(* IEC 61131-3 sources: plc-automation-skill/codesys-st, 4 files *)

(* ---- DUT_CascadeTypes.ST ---- *)
TYPE E_CascadeState :
(
    Stopped := 0,
    SelectLead := 10,
    StartLead := 20,
    RunningCascade := 30,
    StageUp := 40,
    StageDown := 50,
    Tripped := 90
);
END_TYPE

TYPE ST_VSD_Cmd :
STRUCT
    xInhibit : BOOL;
    xRunCmd : BOOL;
    rSpeedRefPct : REAL;
END_STRUCT
END_TYPE

TYPE ST_VSD_Sts :
STRUCT
    xReady : BOOL;
    xRunning : BOOL;
    xFaulted : BOOL;
    xLocal : BOOL;
    xAvailable : BOOL;
    xTripLatched : BOOL;
    xStartFail : BOOL;
    rRuntimeHours : REAL;
    rSpeedFbPct : REAL;
END_STRUCT
END_TYPE

TYPE ST_VSD :
STRUCT
    Cmd : ST_VSD_Cmd;
    Sts : ST_VSD_Sts;
END_STRUCT
END_TYPE

TYPE ST_CascadeCmd :
STRUCT
    xAutoMode : BOOL;
    xManualMode : BOOL;
    xStart : BOOL;
    xStop : BOOL;
    xReset : BOOL;
    xRotateLead : BOOL;
END_STRUCT
END_TYPE

TYPE ST_CascadeCfg :
STRUCT
    iMaxRunning : INT := 5;
    rStageOnSpeedPct : REAL := 90.0;
    rStageOffSpeedPct : REAL := 45.0;
    tStageOnDelay : TIME := T#30S;
    tStageOffDelay : TIME := T#60S;
    tStartTimeout : TIME := T#10S;
    tMinRunTime : TIME := T#120S;
    tMinStopTime : TIME := T#120S;
    rSpeedMinPct : REAL := 0.0;
    rSpeedMaxPct : REAL := 100.0;
END_STRUCT
END_TYPE

TYPE ST_CascadeSts :
STRUCT
    eState : E_CascadeState;
    xAnyTrip : BOOL;
    xPermissiveOK : BOOL;
    iRunningCount : INT;
    iAvailableCount : INT;
    iLeadIndex : INT;
    iNextStageIndex : INT;
    rSpeedDemandPct : REAL;
    xAlarmNoAvailableVSD : BOOL;
    xAlarmStageFail : BOOL;
END_STRUCT
END_TYPE

TYPE ST_Cascade :
STRUCT
    Cmd : ST_CascadeCmd;
    Cfg : ST_CascadeCfg;
    Sts : ST_CascadeSts;
    rPV : REAL;
    rSP : REAL;
    rPIDOutPct : REAL;
END_STRUCT
END_TYPE

(* ---- GVL_IO.ST ---- *)
VAR_GLOBAL
    (* Group control and status. Bind HMI/SCADA tags to CP01 where required. *)
    CP01 : ST_Cascade;

    (* Internal VSD array, indexes 1..5. *)
    CP01_VSD : ARRAY[1..5] OF ST_VSD;

    (* Safety/process permissives mapped from real I/O or safety status. *)
    CP01_xEStopOK : BOOL;
    CP01_xProcessPermissiveOK : BOOL;

    (* Raw VSD inputs. Replace these with mapped fieldbus or I/O addresses. *)
    I_VSD01_xReady : BOOL;
    I_VSD01_xRunning : BOOL;
    I_VSD01_xFaulted : BOOL;
    I_VSD01_xLocal : BOOL;

    I_VSD02_xReady : BOOL;
    I_VSD02_xRunning : BOOL;
    I_VSD02_xFaulted : BOOL;
    I_VSD02_xLocal : BOOL;

    I_VSD03_xReady : BOOL;
    I_VSD03_xRunning : BOOL;
    I_VSD03_xFaulted : BOOL;
    I_VSD03_xLocal : BOOL;

    I_VSD04_xReady : BOOL;
    I_VSD04_xRunning : BOOL;
    I_VSD04_xFaulted : BOOL;
    I_VSD04_xLocal : BOOL;

    I_VSD05_xReady : BOOL;
    I_VSD05_xRunning : BOOL;
    I_VSD05_xFaulted : BOOL;
    I_VSD05_xLocal : BOOL;

    (* Raw VSD outputs. Replace these with mapped fieldbus or I/O addresses. *)
    O_VSD01_xRunCmd : BOOL;
    O_VSD01_rSpeedRefPct : REAL;

    O_VSD02_xRunCmd : BOOL;
    O_VSD02_rSpeedRefPct : REAL;

    O_VSD03_xRunCmd : BOOL;
    O_VSD03_rSpeedRefPct : REAL;

    O_VSD04_xRunCmd : BOOL;
    O_VSD04_rSpeedRefPct : REAL;

    O_VSD05_xRunCmd : BOOL;
    O_VSD05_rSpeedRefPct : REAL;
END_VAR

(* ---- FB_VSD_Cascade5.ST ---- *)
FUNCTION_BLOCK FB_VSD_Cascade5
VAR_INPUT
    xEStopOK : BOOL;
    xProcessPermissiveOK : BOOL;
    stCmd : ST_CascadeCmd;
    stCfg : ST_CascadeCfg;
    rPIDOutPct : REAL;
END_VAR
VAR_IN_OUT
    aVSD : ARRAY[1..5] OF ST_VSD;
END_VAR
VAR_OUTPUT
    stSts : ST_CascadeSts;
END_VAR
VAR
    i : INT;
    iScanIndex : INT;
    iNextLeadIndex : INT := 1;
    xRotateLeadPrev : BOOL;
    tStageOn : TON;
    tStageOff : TON;
    atStartFail : ARRAY[1..5] OF TON;
    atMinRun : ARRAY[1..5] OF TON;
    atMinStop : ARRAY[1..5] OF TON;
    cfg : ST_CascadeCfg;
END_VAR

(* Clamp configuration locally. *)
cfg := stCfg;

IF cfg.iMaxRunning < 1 THEN
    cfg.iMaxRunning := 1;
ELSIF cfg.iMaxRunning > 5 THEN
    cfg.iMaxRunning := 5;
END_IF;

IF cfg.rSpeedMinPct < 0.0 THEN
    cfg.rSpeedMinPct := 0.0;
END_IF;

IF cfg.rSpeedMaxPct > 100.0 THEN
    cfg.rSpeedMaxPct := 100.0;
END_IF;

IF cfg.rSpeedMaxPct < cfg.rSpeedMinPct THEN
    cfg.rSpeedMaxPct := cfg.rSpeedMinPct;
END_IF;

(* Clamp speed demand. PID is normally calculated outside this FB. *)
stSts.rSpeedDemandPct := rPIDOutPct;
IF stSts.rSpeedDemandPct < cfg.rSpeedMinPct THEN
    stSts.rSpeedDemandPct := cfg.rSpeedMinPct;
ELSIF stSts.rSpeedDemandPct > cfg.rSpeedMaxPct THEN
    stSts.rSpeedDemandPct := cfg.rSpeedMaxPct;
END_IF;

(* Group permissive. Reset never starts equipment. *)
stSts.xPermissiveOK :=
    stCmd.xAutoMode AND
    xEStopOK AND
    xProcessPermissiveOK;

stSts.xAnyTrip := (NOT xEStopOK) OR (NOT xProcessPermissiveOK);

(* Rotate preferred lead for next start. *)
IF stCmd.xRotateLead AND NOT xRotateLeadPrev THEN
    iNextLeadIndex := iNextLeadIndex + 1;
    IF iNextLeadIndex > 5 THEN
        iNextLeadIndex := 1;
    END_IF;
END_IF;
xRotateLeadPrev := stCmd.xRotateLead;

IF (iNextLeadIndex < 1) OR (iNextLeadIndex > 5) THEN
    iNextLeadIndex := 1;
END_IF;

(* Per-drive availability, trips, counts, and timers. *)
stSts.iRunningCount := 0;
stSts.iAvailableCount := 0;

FOR i := 1 TO 5 DO
    aVSD[i].Sts.xAvailable :=
        aVSD[i].Sts.xReady AND
        NOT aVSD[i].Sts.xFaulted AND
        NOT aVSD[i].Sts.xLocal AND
        NOT aVSD[i].Cmd.xInhibit AND
        NOT aVSD[i].Sts.xTripLatched;

    IF aVSD[i].Sts.xFaulted OR NOT xEStopOK THEN
        aVSD[i].Sts.xTripLatched := TRUE;
    END_IF;

    IF stCmd.xReset AND NOT aVSD[i].Sts.xFaulted AND xEStopOK THEN
        aVSD[i].Sts.xTripLatched := FALSE;
        aVSD[i].Sts.xStartFail := FALSE;
    END_IF;

    IF aVSD[i].Sts.xTripLatched OR
       aVSD[i].Sts.xFaulted OR
       aVSD[i].Sts.xLocal OR
       aVSD[i].Cmd.xInhibit THEN
        aVSD[i].Cmd.xRunCmd := FALSE;
        aVSD[i].Cmd.rSpeedRefPct := 0.0;
    END_IF;

    IF aVSD[i].Sts.xRunning THEN
        stSts.iRunningCount := stSts.iRunningCount + 1;
    END_IF;

    IF aVSD[i].Sts.xAvailable THEN
        stSts.iAvailableCount := stSts.iAvailableCount + 1;
    END_IF;

    atStartFail[i](IN := aVSD[i].Cmd.xRunCmd AND NOT aVSD[i].Sts.xRunning, PT := cfg.tStartTimeout);
    IF atStartFail[i].Q THEN
        aVSD[i].Sts.xStartFail := TRUE;
        aVSD[i].Sts.xTripLatched := TRUE;
    END_IF;

    atMinRun[i](IN := aVSD[i].Sts.xRunning, PT := cfg.tMinRunTime);
    atMinStop[i](IN := NOT aVSD[i].Sts.xRunning, PT := cfg.tMinStopTime);
END_FOR;

IF stSts.xAnyTrip OR stCmd.xStop THEN
    stSts.eState := E_CascadeState.Stopped;
END_IF;

CASE stSts.eState OF
    E_CascadeState.Stopped:
        FOR i := 1 TO 5 DO
            aVSD[i].Cmd.xRunCmd := FALSE;
            aVSD[i].Cmd.rSpeedRefPct := 0.0;
        END_FOR;

        stSts.xAlarmNoAvailableVSD := FALSE;
        stSts.xAlarmStageFail := FALSE;
        stSts.iLeadIndex := 0;
        stSts.iNextStageIndex := 0;

        IF stCmd.xStart AND stSts.xPermissiveOK THEN
            stSts.eState := E_CascadeState.SelectLead;
        END_IF;

    E_CascadeState.SelectLead:
        stSts.iLeadIndex := 0;

        FOR i := 0 TO 4 DO
            iScanIndex := iNextLeadIndex + i;
            IF iScanIndex > 5 THEN
                iScanIndex := iScanIndex - 5;
            END_IF;

            IF aVSD[iScanIndex].Sts.xAvailable AND atMinStop[iScanIndex].Q THEN
                stSts.iLeadIndex := iScanIndex;
                iNextLeadIndex := stSts.iLeadIndex + 1;
                IF iNextLeadIndex > 5 THEN
                    iNextLeadIndex := 1;
                END_IF;
                EXIT;
            END_IF;
        END_FOR;

        IF stSts.iLeadIndex > 0 THEN
            stSts.eState := E_CascadeState.StartLead;
        ELSE
            stSts.xAlarmNoAvailableVSD := TRUE;
            stSts.eState := E_CascadeState.Tripped;
        END_IF;

    E_CascadeState.StartLead:
        aVSD[stSts.iLeadIndex].Cmd.xRunCmd := TRUE;
        aVSD[stSts.iLeadIndex].Cmd.rSpeedRefPct := stSts.rSpeedDemandPct;

        IF aVSD[stSts.iLeadIndex].Sts.xRunning THEN
            stSts.eState := E_CascadeState.RunningCascade;
        ELSIF NOT stSts.xPermissiveOK THEN
            stSts.eState := E_CascadeState.Stopped;
        END_IF;

    E_CascadeState.RunningCascade:
        FOR i := 1 TO 5 DO
            IF aVSD[i].Cmd.xRunCmd THEN
                aVSD[i].Cmd.rSpeedRefPct := stSts.rSpeedDemandPct;
            ELSE
                aVSD[i].Cmd.rSpeedRefPct := 0.0;
            END_IF;
        END_FOR;

        tStageOn(
            IN := (stSts.rSpeedDemandPct >= cfg.rStageOnSpeedPct) AND
                  (stSts.iRunningCount < cfg.iMaxRunning),
            PT := cfg.tStageOnDelay
        );

        tStageOff(
            IN := (stSts.rSpeedDemandPct <= cfg.rStageOffSpeedPct) AND
                  (stSts.iRunningCount > 1),
            PT := cfg.tStageOffDelay
        );

        IF tStageOn.Q THEN
            stSts.eState := E_CascadeState.StageUp;
        ELSIF tStageOff.Q THEN
            stSts.eState := E_CascadeState.StageDown;
        END_IF;

    E_CascadeState.StageUp:
        stSts.iNextStageIndex := 0;

        FOR i := 1 TO 5 DO
            iScanIndex := stSts.iLeadIndex + i;
            IF iScanIndex > 5 THEN
                iScanIndex := iScanIndex - 5;
            END_IF;

            IF aVSD[iScanIndex].Sts.xAvailable AND
               NOT aVSD[iScanIndex].Cmd.xRunCmd AND
               atMinStop[iScanIndex].Q THEN
                stSts.iNextStageIndex := iScanIndex;
                EXIT;
            END_IF;
        END_FOR;

        IF stSts.iNextStageIndex > 0 THEN
            aVSD[stSts.iNextStageIndex].Cmd.xRunCmd := TRUE;
            aVSD[stSts.iNextStageIndex].Cmd.rSpeedRefPct := stSts.rSpeedDemandPct;
        ELSE
            stSts.xAlarmStageFail := TRUE;
        END_IF;

        tStageOn(IN := FALSE, PT := cfg.tStageOnDelay);
        stSts.eState := E_CascadeState.RunningCascade;

    E_CascadeState.StageDown:
        stSts.iNextStageIndex := 0;

        FOR i := 5 TO 1 BY -1 DO
            iScanIndex := stSts.iLeadIndex + i - 1;
            IF iScanIndex > 5 THEN
                iScanIndex := iScanIndex - 5;
            END_IF;

            IF (iScanIndex <> stSts.iLeadIndex) AND
               aVSD[iScanIndex].Cmd.xRunCmd AND
               atMinRun[iScanIndex].Q THEN
                stSts.iNextStageIndex := iScanIndex;
                EXIT;
            END_IF;
        END_FOR;

        IF stSts.iNextStageIndex > 0 THEN
            aVSD[stSts.iNextStageIndex].Cmd.xRunCmd := FALSE;
            aVSD[stSts.iNextStageIndex].Cmd.rSpeedRefPct := 0.0;
        END_IF;

        tStageOff(IN := FALSE, PT := cfg.tStageOffDelay);
        stSts.eState := E_CascadeState.RunningCascade;

    E_CascadeState.Tripped:
        FOR i := 1 TO 5 DO
            aVSD[i].Cmd.xRunCmd := FALSE;
            aVSD[i].Cmd.rSpeedRefPct := 0.0;
        END_FOR;

        IF stCmd.xReset AND NOT stSts.xAnyTrip THEN
            stSts.eState := E_CascadeState.Stopped;
        END_IF;

ELSE
    stSts.eState := E_CascadeState.Tripped;
END_CASE;

(* ---- PRG_Main.ST ---- *)
PROGRAM PRG_Main
VAR
    fbCascade : FB_VSD_Cascade5;
END_VAR

(* Map raw inputs into the internal VSD structures. *)
CP01_VSD[1].Sts.xReady := I_VSD01_xReady;
CP01_VSD[1].Sts.xRunning := I_VSD01_xRunning;
CP01_VSD[1].Sts.xFaulted := I_VSD01_xFaulted;
CP01_VSD[1].Sts.xLocal := I_VSD01_xLocal;

CP01_VSD[2].Sts.xReady := I_VSD02_xReady;
CP01_VSD[2].Sts.xRunning := I_VSD02_xRunning;
CP01_VSD[2].Sts.xFaulted := I_VSD02_xFaulted;
CP01_VSD[2].Sts.xLocal := I_VSD02_xLocal;

CP01_VSD[3].Sts.xReady := I_VSD03_xReady;
CP01_VSD[3].Sts.xRunning := I_VSD03_xRunning;
CP01_VSD[3].Sts.xFaulted := I_VSD03_xFaulted;
CP01_VSD[3].Sts.xLocal := I_VSD03_xLocal;

CP01_VSD[4].Sts.xReady := I_VSD04_xReady;
CP01_VSD[4].Sts.xRunning := I_VSD04_xRunning;
CP01_VSD[4].Sts.xFaulted := I_VSD04_xFaulted;
CP01_VSD[4].Sts.xLocal := I_VSD04_xLocal;

CP01_VSD[5].Sts.xReady := I_VSD05_xReady;
CP01_VSD[5].Sts.xRunning := I_VSD05_xRunning;
CP01_VSD[5].Sts.xFaulted := I_VSD05_xFaulted;
CP01_VSD[5].Sts.xLocal := I_VSD05_xLocal;

(* Cascade control. CP01.rPIDOutPct should come from a CODESYS PID/PID_FIXCYCLE loop or external demand calculation. *)
fbCascade(
    xEStopOK := CP01_xEStopOK,
    xProcessPermissiveOK := CP01_xProcessPermissiveOK,
    stCmd := CP01.Cmd,
    stCfg := CP01.Cfg,
    rPIDOutPct := CP01.rPIDOutPct,
    aVSD := CP01_VSD,
    stSts => CP01.Sts
);

(* Map internal commands to raw outputs. *)
O_VSD01_xRunCmd := CP01_VSD[1].Cmd.xRunCmd;
O_VSD01_rSpeedRefPct := CP01_VSD[1].Cmd.rSpeedRefPct;

O_VSD02_xRunCmd := CP01_VSD[2].Cmd.xRunCmd;
O_VSD02_rSpeedRefPct := CP01_VSD[2].Cmd.rSpeedRefPct;

O_VSD03_xRunCmd := CP01_VSD[3].Cmd.xRunCmd;
O_VSD03_rSpeedRefPct := CP01_VSD[3].Cmd.rSpeedRefPct;

O_VSD04_xRunCmd := CP01_VSD[4].Cmd.xRunCmd;
O_VSD04_rSpeedRefPct := CP01_VSD[4].Cmd.rSpeedRefPct;

O_VSD05_xRunCmd := CP01_VSD[5].Cmd.xRunCmd;
O_VSD05_rSpeedRefPct := CP01_VSD[5].Cmd.rSpeedRefPct;
